PROGRAM Safety

END_PROGRAM

(* stored: Version 1.1.0.1
   POU Safety: Id {c0fa21ec-79d9-432e-a6c8-9a56af19668a}, SpecialFunc None *)
